(* IEC 61131-3 sources: programs/VI-54/VI-54_20171205/VI-54_20171205/Stations/Screen/LseClass170718/Class/DiagnosticStation_PLC, 1 file *)

(* ---- DiagnosticStation_PLC.st ---- *)
(*!
<Class
	Name               = "DiagnosticStation_PLC"
	Revision           = "1.1"
	RealtimeTask       = "false"
	CyclicTask         = "false"
	BackgroundTask     = "false"
	Sigmatek           = "false"
	OSInterface        = "false"
	HighPriority       = "false"
	Automatic          = "false"
	UpdateMode         = "Prescan"
	SharedCommandTable = "true"
	Objectsize         = "(960,360)"
	Comment            = "Use this class as station for the diagnostic export.">
	<Channels>
		<Server Name="ClassSvr" Visualized="false" Initialize="false" WriteProtected="true" Retentive="false"/>
		<Server Name="ID_Destination" Visualized="false" Initialize="true" WriteProtected="true" Retentive="false"/>
		<Server Name="ID_Source" Visualized="false" Initialize="true" WriteProtected="true" Retentive="false"/>
		<Client Name="cPrio" Required="true" Internal="false" Comment="Communication priority number."/>
		<Client Name="cUserFunction" Required="true" Internal="false" Comment="Object channel to DiagnosticUserFunction_PLC."/>
		<Client Name="DiagnosticWork_PLC" Required="true" Internal="true"/>
		<Client Name="ReceiveDataCMD_PLC" Required="true" Internal="true"/>
		<Client Name="SendDataCMD_PLC" Required="true" Internal="true"/>
		<Client Name="toDataManager" Required="true" Internal="false" Comment="Connection to communication data manager."/>
	</Channels>
	<RevDoku>
		<Owner Company="Sigmatek"/>
		<Dokumentation Revision="1.1" Date="2016-06-15" Author="HasHan" Company="Sigmatek" Description="changes at the inside"/>
		<Dokumentation Revision="1.0" Date="2016-06-02" Author="HötAnt" Company="Sigmatek" Description="Creation"/>
	</RevDoku>
	<Network Name="DiagnosticStation_PLC">
		<!-- List of Components in this network -->
		<Components>
			<Object
				Name           = "DiagnosticWork_PLC"
				Class          = "DiagnosticWork_PLC"
				Position       = "(420,690)"
				Visualized     = "false"
				BackgroundTime = "2 ms">
				<Channels>
					<Server Name="sStatus"/>
					<Client Name="cToCom"/>
					<Client Name="cUserFunction"/>
				</Channels>
			</Object>
			<Object
				Name       = "ReceiveDataCMD_PLC"
				Class      = "ReceiveDataCMD_PLC"
				Position   = "(1080,510)"
				Visualized = "false">
				<Channels>
					<Server Name="ClassSvr"/>
					<Server Name="ID_Source"/>
					<Server Name="sRecvCnt"/>
					<Client Name="cDiagnosticWork_PLC"/>
					<Client Name="toDataManager"/>
				</Channels>
			</Object>
			<Object
				Name       = "SendDataCMD_PLC"
				Class      = "SendDataCMD_PLC"
				Position   = "(450,120)"
				Visualized = "false">
				<Channels>
					<Server Name="ClassSvr"/>
					<Server Name="ID_Destination"/>
					<Server Name="ID_Source"/>
					<Server Name="sSendCnt"/>
					<Server Name="sSendErr"/>
					<Client Name="cPrio"/>
					<Client Name="cStation"/>
					<Client Name="toDataManager"/>
				</Channels>
			</Object>
		</Components>
		<Comments>
		</Comments>
		<!-- List of Connections in this network -->
		<Connections>
			<Connection Source="this.DiagnosticWork_PLC" Destination="DiagnosticWork_PLC.sStatus"/>
			<Connection Source="this.ID_Source" Destination="SendDataCMD_PLC.ID_Source" Vertices="(1944,270),(952,330),"/>
			<Connection Source="this.ID_Destination" Destination="SendDataCMD_PLC.ID_Destination" Vertices="(1944,330),(952,270),"/>
			<Connection Source="DiagnosticWork_PLC.cToCom" Destination="SendDataCMD_PLC.ClassSvr" Vertices="(420,840),(952,210),"/>
			<Connection Source="DiagnosticWork_PLC.cUserFunction" Destination="this.cUserFunction" Vertices="(420,780),(38,270),"/>
			<Connection Source="this.SendDataCMD_PLC" Destination="SendDataCMD_PLC.ClassSvr"/>
			<Connection Source="SendDataCMD_PLC.cStation" Destination="DiagnosticWork_PLC.sStatus" Vertices="(450,330),(914,780),"/>
			<Connection Source="SendDataCMD_PLC.cPrio" Destination="this.cPrio" Vertices="(450,270),(360,270),(360,330),(38,330),"/>
			<Connection Source="this.ReceiveDataCMD_PLC" Destination="ReceiveDataCMD_PLC.ClassSvr"/>
			<Connection Source="ReceiveDataCMD_PLC.cDiagnosticWork_PLC" Destination="DiagnosticWork_PLC.sStatus" Vertices="(1080,660),(914,780),"/>
			<Connection Source="ReceiveDataCMD_PLC.toDataManager" Destination="this.toDataManager" Vertices="(1080,600),(270,600),(270,210),(38,210),"/>
			<Connection Source="SendDataCMD_PLC.toDataManager" Destination="this.toDataManager" Vertices="(450,210),(38,210),"/>
		</Connections>
		<!-- Headerfiles -->
		<Options>
		</Options>
	</Network>
</Class>
*)
DiagnosticStation_PLC : CLASS
  //Servers:
	ClassSvr 	: SvrChCmd_DINT;
	ID_Source 	: SvrCh_DINT;
	ID_Destination 	: SvrCh_DINT;
  //Clients:
	DiagnosticWork_PLC 	: CltChCmd_DiagnosticWork_PLC;
	toDataManager 	: CltChCmd_DataManager;
	cUserFunction 	: CltChCmd_DiagnosticUserFunction_PLC;
	cPrio 	: CltCh_DINT;
	SendDataCMD_PLC 	: CltChCmd_SendDataCMD_PLC;
	ReceiveDataCMD_PLC 	: CltChCmd_ReceiveDataCMD_PLC;
  //Variables:
  //Functions:

	FUNCTION VIRTUAL GLOBAL Init;

	FUNCTION VIRTUAL GLOBAL ID_Source::Read
		VAR_OUTPUT
			output (EAX) 	: DINT;
		END_VAR;

	FUNCTION VIRTUAL GLOBAL ID_Destination::Read
		VAR_OUTPUT
			output (EAX) 	: DINT;
		END_VAR;
  //Tables:
	FUNCTION @STD
		VAR_OUTPUT
			ret_code	: CONFSTATES;
		END_VAR;
	FUNCTION GLOBAL TAB @CT_;
END_CLASS;

#pragma using DiagnosticWork_PLC
#pragma using ReceiveDataCMD_PLC
#pragma using SendDataCMD_PLC
#pragma usingLtd DataManager
#pragma usingLtd DiagnosticUserFunction_PLC

FUNCTION VIRTUAL GLOBAL DiagnosticStation_PLC::Init

  if _FirstScan then
    ReceiveDataCMD_PLC.ID_Source := ID_Source; //set the same ID to the receive-object
  end_if;

END_FUNCTION

FUNCTION VIRTUAL GLOBAL DiagnosticStation_PLC::ID_Source::Read
	VAR_OUTPUT
		output (EAX) 	: DINT;
	END_VAR

	ID_Source := SendDataCMD_PLC.ID_Source.Read();
	output := ID_Source;

END_FUNCTION

FUNCTION VIRTUAL GLOBAL DiagnosticStation_PLC::ID_Destination::Read
	VAR_OUTPUT
		output (EAX) 	: DINT;
	END_VAR

	ID_Destination := SendDataCMD_PLC.ID_Destination.Read();
	output := ID_Destination;

END_FUNCTION
